; ANGLE 51.0 (Not valid for Circ layers and non-tubes)
$APO.CDIS=85
$VEL_EXTAX[1]=100
FOR N_CYC=1 to 26
 LIN_REL {X  -1.263,Y -17.738,A +0.664,E1 +5.909,E3 +39.726,E4 +39.726} C_DIS
 LIN_REL {X  -1.207,Y -17.519,A +6.151,E1 +1.101,E3 +33.522,E4 +33.522} C_DIS
 LIN_REL {X  +0.132,Y -25.137,A +10.003,E1 -0.421,E3 +50.269,E4 +50.269} C_DIS
 LIN_REL {X  +1.938,Y -24.469,A +9.586,E1 -2.860,E3 +55.196,E4 +55.196} C_DIS
 LIN_REL {X  +1.088,Y -27.792,A +3.019,E1 -0.955,E3 +68.896,E4 +68.896} C_DIS
 LIN_REL {X  -1.412,Y -27.938,A +0.462,E1 -0.637,E3 +74.120,E4 +74.120} C_DIS
 LIN_REL {X  -1.550,Y -28.084,A +0.079,E1 -0.824,E3 +75.675,E4 +75.675} C_DIS
 LIN_REL {X  -0.218,Y -37.855,A +0.031,E1 +0.120,E3 +99.590,E4 +99.590} C_DIS
 LIN_REL {X  +0.045,Y -439.757,A +0.006,E1 -0.006,E3 +1160.946,E4 +1160.946} C_DIS
 LIN_REL {X  -0.042,Y -41.169,A +0.005,E1 -0.034,E3 +108.768,E4 +108.768} C_DIS
 LIN_REL {X  +1.080,Y -35.595,A +0.045,E1 +0.289,E3 +92.600,E4 +92.600} C_DIS
 LIN_REL {X  +3.273,Y -34.380,A +0.217,E1 +0.416,E3 +91.278,E4 +91.278} C_DIS
 LIN_REL {X  +2.743,Y -26.470,A +1.240,E1 -2.201,E3 +76.331,E4 +76.331} C_DIS
 LIN_REL {X  +2.631,Y -16.478,A +6.378,E1 -6.830,E3 +59.126,E4 +59.126} C_DIS
 LIN_REL {X  +2.229,Y -8.399,A +11.491,E1 -13.235,E3 +51.842,E4 +51.842} C_DIS
 LIN_REL {X  +0.487,Y -0.700,A +8.521,E1 -13.721,E3 +42.558,E4 +42.558} C_DIS
 LIN_REL {X  -1.738,Y +4.804,A +2.101,E1 -9.621,E3 +38.319,E4 +38.319} C_DIS
 LIN_REL {X  -4.726,Y +16.117,A +0.001,E1 -12.271,E3 +54.688,E4 +54.688} C_DIS
 LIN_REL {X  -3.801,Y +19.459,A -0.092,E1 -8.574,E3 +43.826,E4 +43.826} C_DIS
 LIN_REL {X  -1.602,Y +15.638,A -4.416,E1 -2.235,E3 +29.939,E4 +29.939} C_DIS
 LIN_REL {X  -0.782,Y +22.587,A -8.423,E1 -0.320,E3 +44.108,E4 +44.108} C_DIS
 LIN_REL {X  +1.659,Y +27.200,A -11.255,E1 +2.496,E3 +59.206,E4 +59.206} C_DIS
 LIN_REL {X  +1.774,Y +29.070,A -4.803,E1 +1.404,E3 +70.515,E4 +70.515} C_DIS
 LIN_REL {X  -1.281,Y +30.779,A -0.863,E1 +0.755,E3 +80.640,E4 +80.640} C_DIS
 LIN_REL {X  -1.562,Y +27.869,A -0.109,E1 +1.005,E3 +75.559,E4 +75.559} C_DIS
 LIN_REL {X  -0.402,Y +34.896,A -0.035,E1 -0.167,E3 +91.664,E4 +91.664} C_DIS
 LIN_REL {X  +0.061,Y +446.163,A -0.005,E1 +0.005,E3 +1177.603,E4 +1177.603} C_DIS
 LIN_REL {X  -0.041,Y +41.178,A -0.009,E1 +0.036,E3 +108.772,E4 +108.772} C_DIS
 LIN_REL {X  +1.058,Y +35.617,A -0.046,E1 -0.293,E3 +92.627,E4 +92.627} C_DIS
 LIN_REL {X  +3.023,Y +32.120,A -0.168,E1 -0.412,E3 +85.081,E4 +85.081} C_DIS
 LIN_REL {X  +2.606,Y +25.937,A -0.789,E1 +1.529,E3 +73.528,E4 +73.528} C_DIS
 LIN_REL {X  +2.648,Y +17.147,A -4.931,E1 +5.567,E3 +58.465,E4 +58.465} C_DIS
 LIN_REL {X  +2.311,Y +9.487,A -12.018,E1 +12.736,E3 +50.262,E4 +50.262} C_DIS
 LIN_REL {X  +0.814,Y +2.053,A -9.484,E1 +14.819,E3 +47.597,E4 +47.597} C_DIS
 LIN_REL {X  -1.900,Y -4.606,A -2.553,E1 +10.763,E3 +43.244,E4 +43.244} C_DIS
 LIN_REL {X  -4.922,Y -13.188,A -0.001,E1 +10.333,E3 +35.563,E4 +35.563} C_DIS
 LIN_REL {X  -3.151,Y -10.847,A -0.000,E1 +6.334,E3 +35.274,E4 +35.274} C_DIS
ENDFOR

HALT
LIN {X -171.700,Y 1348.990,Z 0.000,A -27.171, B 0.00, C 0.00,E1 30.065}
HALT

; PLY 29 OF 41 (Connector)

; ANGLE 51.0 (Not valid for Circ layers and non-tubes)
$APO.CDIS=85
$VEL_EXTAX[1]=100
FOR N_CYC=1 to 1
 LIN_REL {X  +0.000,Y -9.233,A +0.373,E1 +2.358,E3 +17.818,E4 +17.818} C_DIS
 LIN_REL {X  +0.000,Y -13.860,A -0.779,E1 +4.453,E3 +24.815,E4 +24.815} C_DIS
 LIN_REL {X  +0.000,Y -18.793,A +5.783,E1 +1.657,E3 +30.501,E4 +30.501} C_DIS
 LIN_REL {X  +0.000,Y -28.514,A +11.207,E1 -0.369,E3 +47.105,E4 +47.105} C_DIS
 LIN_REL {X  +0.000,Y -29.574,A +8.105,E1 -0.986,E3 +52.158,E4 +52.158} C_DIS
 LIN_REL {X  +0.000,Y -39.267,A +2.075,E1 +1.140,E3 +70.967,E4 +70.967} C_DIS
 LIN_REL {X  +0.000,Y -46.416,A +0.339,E1 +1.591,E3 +81.647,E4 +81.647} C_DIS
 LIN_REL {X  +0.000,Y -56.639,A +0.061,E1 +2.018,E3 +93.300,E4 +93.300} C_DIS
 LIN_REL {X  +0.000,Y -63.527,A +0.007,E1 +2.194,E3 +97.039,E4 +97.039} C_DIS
 LIN_REL {X  +0.000,Y -66.959,A +0.000,E1 +2.174,E3 +94.666,E4 +94.666} C_DIS
 LIN_REL {X  +0.000,Y -70.250,A +0.000,E1 +2.135,E3 +91.980,E4 +91.980} C_DIS
 LIN_REL {X  +0.000,Y -70.396,A +0.000,E1 +2.009,E3 +85.511,E4 +85.511} C_DIS
 LIN_REL {X  +0.000,Y -73.804,A +0.000,E1 +1.984,E3 +83.251,E4 +83.251} C_DIS
 LIN_REL {X  +0.000,Y -77.291,A +0.000,E1 +1.961,E3 +80.882,E4 +80.882} C_DIS
 LIN_REL {X  +0.000,Y -77.374,A +0.002,E1 +1.847,E3 +75.125,E4 +75.125} C_DIS
 LIN_REL {X  +0.000,Y -70.709,A +0.068,E1 +1.551,E3 +64.105,E4 +64.105} C_DIS
 LIN_REL {X  +0.000,Y -55.789,A +0.709,E1 +0.995,E3 +48.959,E4 +48.959} C_DIS
 LIN_REL {X  +0.000,Y -40.604,A +4.575,E1 -1.183,E3 +41.358,E4 +41.358} C_DIS
 LIN_REL {X  +0.000,Y -25.454,A +10.692,E1 -5.269,E3 +34.062,E4 +34.062} C_DIS
 LIN_REL {X  +0.000,Y -12.708,A +10.798,E1 -8.471,E3 +24.267,E4 +24.267} C_DIS
 LIN_REL {X  +0.000,Y -7.379,A +3.152,E1 -5.505,E3 +25.747,E4 +25.747} C_DIS
 LIN_REL {X  +0.000,Y +0.970,A +0.004,E1 -4.558,E3 +33.819,E4 +33.819} C_DIS
 LIN_REL {X  +0.000,Y +10.934,A +0.000,E1 -10.007,E3 +28.863,E4 +28.863} C_DIS
 LIN_REL {X  +0.000,Y +19.588,A +0.000,E1 -13.423,E3 +28.165,E4 +28.165} C_DIS
 LIN_REL {X  +0.000,Y +12.206,A +0.000,E1 -10.399,E3 +11.631,E4 +11.631} C_DIS
 LIN_REL {X  +0.000,Y +1.140,A +0.000,E1 +0.761,E3 +0.965,E4 +0.965} C_DIS
 LIN_REL {X  +0.000,Y +3.435,A +0.000,E1 +4.724,E3 +3.121,E4 +3.121} C_DIS
 LIN_REL {X  +0.000,Y +16.386,A +0.000,E1 -14.565,E3 +13.019,E4 +13.019} C_DIS
 LIN_REL {X  +0.000,Y +31.237,A +0.000,E1 -16.911,E3 +19.850,E4 +19.850} C_DIS
 LIN_REL {X  +0.000,Y +24.263,A +0.000,E1 -12.079,E3 +15.482,E4 +15.482} C_DIS
ENDFOR

HALT
LIN {X -157.685,Y 535.549,Z 0.000,A 30.000, B 0.00, C 0.00,E1 -43.006}
HALT

; PLY 30 OF 41 (Helical)

; ANGLE 51.0 (Not valid for Circ layers and non-tubes)
$APO.CDIS=85
$VEL_EXTAX[1]=100
FOR N_CYC=1 to 49
 LIN_REL {X  -9.992,Y +38.440,A +0.000,E1 -12.506,E3 +27.076,E4 +27.076} C_DIS
 LIN_REL {X  -2.820,Y +34.329,A -0.140,E1 -4.875,E3 +21.050,E4 +21.050} C_DIS
 LIN_REL {X  -0.513,Y +17.919,A -5.095,E1 +0.029,E3 +11.726,E4 +11.726} C_DIS
 LIN_REL {X  -0.353,Y +14.948,A -0.644,E1 -0.565,E3 +10.215,E4 +10.215} C_DIS
 LIN_REL {X  -0.076,Y +14.598,A -1.861,E1 -0.455,E3 +10.433,E4 +10.433} C_DIS
 LIN_REL {X  +0.253,Y +25.054,A -7.468,E1 +0.260,E3 +18.780,E4 +18.780} C_DIS
 LIN_REL {X  +0.495,Y +39.543,A -9.068,E1 +0.940,E3 +31.936,E4 +31.936} C_DIS
 LIN_REL {X  +0.350,Y +52.493,A -5.061,E1 +0.537,E3 +46.398,E4 +46.398} C_DIS
 LIN_REL {X  +0.714,Y +65.315,A -0.637,E1 -0.061,E3 +60.775,E4 +60.775} C_DIS
 LIN_REL {X  +0.354,Y +72.797,A -0.026,E1 +0.019,E3 +68.477,E4 +68.477} C_DIS
 LIN_REL {X  +0.057,Y +276.942,A -0.000,E1 +0.012,E3 +261.192,E4 +261.192} C_DIS
 LIN_REL {X  +0.037,Y +57.440,A -0.000,E1 +0.014,E3 +54.220,E4 +54.220} C_DIS
 LIN_REL {X  +0.274,Y +42.150,A -0.000,E1 +0.085,E3 +40.041,E4 +40.041} C_DIS
 LIN_REL {X  +0.902,Y +29.530,A -0.002,E1 +0.226,E3 +28.682,E4 +28.682} C_DIS
 LIN_REL {X  +1.263,Y +17.565,A -0.005,E1 +0.283,E3 +17.684,E4 +17.684} C_DIS
 LIN_REL {X  +3.157,Y +23.364,A -0.024,E1 +0.665,E3 +24.764,E4 +24.764} C_DIS
 LIN_REL {X  +9.310,Y +31.543,A -0.347,E1 +1.862,E3 +37.286,E4 +37.286} C_DIS
 LIN_REL {X  +12.432,Y +18.699,A -3.734,E1 +3.126,E3 +27.471,E4 +27.471} C_DIS
 LIN_REL {X  +13.471,Y +12.237,A -11.704,E1 +6.647,E3 +27.002,E4 +27.002} C_DIS
 LIN_REL {X  +8.296,Y +6.142,A -8.436,E1 +5.968,E3 +20.449,E4 +20.449} C_DIS
 LIN_REL {X  +6.939,Y +4.164,A -2.979,E1 +4.722,E3 +22.940,E4 +22.940} C_DIS
 LIN_REL {X  +6.923,Y +3.493,A -2.751,E1 +10.488,E3 +42.442,E4 +42.442} C_DIS
 LIN_REL {X  -1.399,Y -0.415,A -0.018,E1 +13.616,E3 +55.399,E4 +55.399} C_DIS
 LIN_REL {X  -10.123,Y -6.481,A +0.000,E1 +15.056,E3 +45.794,E4 +45.794} C_DIS
 LIN_REL {X  -18.030,Y -13.565,A +0.000,E1 +18.431,E3 +41.692,E4 +41.692} C_DIS
 LIN_REL {X  -18.339,Y -23.904,A +0.000,E1 +18.670,E3 +32.802,E4 +32.802} C_DIS
 LIN_REL {X  -11.143,Y -31.247,A +0.000,E1 +12.210,E3 +24.387,E4 +24.387} C_DIS
 LIN_REL {X  -4.894,Y -37.209,A +0.000,E1 +7.145,E3 +22.801,E4 +22.801} C_DIS
 LIN_REL {X  -0.708,Y -20.875,A +2.543,E1 +0.987,E3 +13.371,E4 +13.371} C_DIS
 LIN_REL {X  -0.360,Y -13.653,A +4.268,E1 -0.155,E3 +9.150,E4 +9.150} C_DIS
 LIN_REL {X  -0.243,Y -17.021,A -0.267,E1 +0.899,E3 +11.930,E4 +11.930} C_DIS
 LIN_REL {X  +0.170,Y -22.146,A +6.338,E1 -0.020,E3 +16.273,E4 +16.273} C_DIS
 LIN_REL {X  +0.520,Y -34.300,A +8.556,E1 -0.682,E3 +26.945,E4 +26.945} C_DIS
 LIN_REL {X  +0.275,Y -48.825,A +7.263,E1 -0.966,E3 +42.019,E4 +42.019} C_DIS
 LIN_REL {X  +0.615,Y -59.709,A +1.212,E1 +0.086,E3 +55.054,E4 +55.054} C_DIS
 LIN_REL {X  +0.533,Y -71.084,A +0.084,E1 -0.000,E3 +66.733,E4 +66.733} C_DIS
 LIN_REL {X  +0.122,Y -305.348,A +0.003,E1 -0.022,E3 +287.956,E4 +287.956} C_DIS
 LIN_REL {X  +0.045,Y -57.401,A +0.000,E1 -0.017,E3 +54.194,E4 +54.194} C_DIS
 LIN_REL {X  +0.339,Y -41.950,A +0.000,E1 -0.101,E3 +39.910,E4 +39.910} C_DIS
 LIN_REL {X  +1.030,Y -29.366,A +0.002,E1 -0.250,E3 +28.637,E4 +28.637} C_DIS
 LIN_REL {X  +1.070,Y -14.362,A +0.003,E1 -0.238,E3 +14.492,E4 +14.492} C_DIS
 LIN_REL {X  +2.587,Y -20.443,A +0.016,E1 -0.547,E3 +21.523,E4 +21.523} C_DIS
 LIN_REL {X  +7.682,Y -29.414,A +0.236,E1 -1.546,E3 +34.044,E4 +34.044} C_DIS
 LIN_REL {X  +11.916,Y -20.738,A +2.572,E1 -2.756,E3 +28.891,E4 +28.891} C_DIS
 LIN_REL {X  +13.331,Y -12.978,A +10.132,E1 -5.754,E3 +26.094,E4 +26.094} C_DIS
 LIN_REL {X  +10.908,Y -8.239,A +10.945,E1 -7.427,E3 +25.783,E4 +25.783} C_DIS
 LIN_REL {X  +8.205,Y -4.895,A +3.479,E1 -5.602,E3 +27.304,E4 +27.304} C_DIS
 LIN_REL {X  +5.935,Y -2.966,A +2.598,E1 -9.964,E3 +39.224,E4 +39.224} C_DIS
 LIN_REL {X  -1.496,Y +0.449,A +0.017,E1 -13.553,E3 +55.117,E4 +55.117} C_DIS
 LIN_REL {X  -10.127,Y +6.477,A +0.000,E1 -14.993,E3 +45.594,E4 +45.594} C_DIS
 LIN_REL {X  -17.619,Y +12.986,A +0.000,E1 -18.049,E3 +40.676,E4 +40.676} C_DIS
 LIN_REL {X  -22.275,Y +29.917,A +0.000,E1 -21.879,E3 +38.845,E4 +38.845} C_DIS
ENDFOR

HALT
LIN {X -172.144,Y 529.033,Z 0.000,A 30.000, B 0.00, C 0.00,E1 -44.225}
HALT

; PLY 31 OF 41 (Connector)

; ANGLE 51.0 (Not valid for Circ layers and non-tubes)
$APO.CDIS=85
$VEL_EXTAX[1]=100
FOR N_CYC=1 to 1
 LIN_REL {X  +0.000,Y +14.319,A +0.000,E1 -4.145,E3 +12.342,E4 +12.342} C_DIS
 LIN_REL {X  +0.000,Y +6.169,A +0.000,E1 -1.493,E3 +5.195,E4 +5.195} C_DIS
 LIN_REL {X  +0.000,Y +13.714,A +0.000,E1 -3.208,E3 +10.742,E4 +10.742} C_DIS
 LIN_REL {X  +0.000,Y +36.143,A -0.001,E1 -5.463,E3 +24.130,E4 +24.130} C_DIS
 LIN_REL {X  +0.000,Y +26.736,A -3.446,E1 -0.505,E3 +19.551,E4 +19.551} C_DIS
 LIN_REL {X  +0.000,Y +25.698,A -6.360,E1 +0.299,E3 +22.076,E4 +22.076} C_DIS
 LIN_REL {X  +0.000,Y +35.270,A -10.863,E1 +1.539,E3 +33.206,E4 +33.206} C_DIS
 LIN_REL {X  +0.000,Y +38.420,A -7.659,E1 +2.559,E3 +44.300,E4 +44.300} C_DIS
 LIN_REL {X  +0.000,Y +44.211,A -1.519,E1 +1.891,E3 +58.868,E4 +58.868} C_DIS
 LIN_REL {X  +0.000,Y +49.956,A -0.142,E1 +1.911,E3 +70.742,E4 +70.742} C_DIS
 LIN_REL {X  +0.000,Y +56.506,A -0.010,E1 +2.198,E3 +85.749,E4 +85.749} C_DIS
 LIN_REL {X  +0.000,Y +61.033,A +0.000,E1 +2.498,E3 +100.307,E4 +100.307} C_DIS
 LIN_REL {X  +0.000,Y +58.632,A +0.000,E1 +2.584,E3 +105.218,E4 +105.218} C_DIS
 LIN_REL {X  +0.000,Y +53.534,A -0.000,E1 +2.555,E3 +105.199,E4 +105.199} C_DIS
 LIN_REL {X  +0.000,Y +41.233,A -0.000,E1 +2.127,E3 +88.197,E4 +88.197} C_DIS
 LIN_REL {X  +0.000,Y +31.694,A -0.000,E1 +1.788,E3 +72.960,E4 +72.960} C_DIS
 LIN_REL {X  +0.000,Y +22.339,A -0.000,E1 +1.883,E3 +54.647,E4 +54.647} C_DIS
 LIN_REL {X  +0.000,Y +12.026,A -0.000,E1 +1.596,E3 +30.477,E4 +30.477} C_DIS
 LIN_REL {X  +0.000,Y +8.605,A -0.000,E1 +0.479,E3 +23.899,E4 +23.899} C_DIS
 LIN_REL {X  +0.000,Y +17.185,A -0.000,E1 +0.297,E3 +43.997,E4 +43.997} C_DIS
 LIN_REL {X  +0.000,Y +22.397,A -0.002,E1 +1.554,E3 +63.484,E4 +63.484} C_DIS
 LIN_REL {X  +0.000,Y +26.340,A -0.006,E1 +1.986,E3 +80.445,E4 +80.445} C_DIS
 LIN_REL {X  +0.000,Y +29.797,A -0.026,E1 +2.502,E3 +100.345,E4 +100.345} C_DIS
 LIN_REL {X  +0.000,Y +26.761,A -0.089,E1 +2.608,E3 +101.540,E4 +101.540} C_DIS
 LIN_REL {X  +0.000,Y +19.332,A -0.202,E1 +2.288,E3 +83.045,E4 +83.045} C_DIS
 LIN_REL {X  +0.000,Y +13.522,A -0.387,E1 +2.080,E3 +65.819,E4 +65.819} C_DIS
 LIN_REL {X  +0.000,Y +9.350,A -0.577,E1 +1.526,E3 +48.552,E4 +48.552} C_DIS
 LIN_REL {X  +0.000,Y +7.090,A -1.004,E1 +0.962,E3 +34.729,E4 +34.729} C_DIS
 LIN_REL {X  +0.000,Y +4.780,A -0.977,E1 +1.016,E3 +28.901,E4 +28.901} C_DIS
 LIN_REL {X  +0.000,Y +4.146,A -1.612,E1 +2.199,E3 +25.934,E4 +25.934} C_DIS
 LIN_REL {X  +0.000,Y +5.726,A -4.369,E1 +5.416,E3 +44.520,E4 +44.520} C_DIS
 LIN_REL {X  +0.000,Y +2.416,A -7.629,E1 +11.123,E3 +57.450,E4 +57.450} C_DIS
 LIN_REL {X  +0.000,Y -2.383,A -3.896,E1 +8.270,E3 +42.248,E4 +42.248} C_DIS
 LIN_REL {X  +0.000,Y -1.687,A -0.589,E1 +2.742,E3 +18.919,E4 +18.919} C_DIS
ENDFOR

HALT
LIN {X -169.560,Y 1333.646,Z 0.000,A -22.240, B 0.00, C 0.00,E1 22.754}
HALT

; PLY 32 OF 41 (Helical)

; ANGLE 51.0 (Not valid for Circ layers and non-tubes)
$APO.CDIS=85
$VEL_EXTAX[1]=100
FOR N_CYC=1 to 16
 LIN_REL {X  +3.047,Y -12.617,A +5.110,E1 +1.887,E3 +50.457,E4 +50.457} C_DIS
 LIN_REL {X  +0.960,Y -17.440,A +9.214,E1 -2.081,E3 +64.163,E4 +64.163} C_DIS
 LIN_REL {X  -1.414,Y -14.583,A +4.594,E1 -1.524,E3 +56.231,E4 +56.231} C_DIS
 LIN_REL {X  -1.370,Y -15.018,A +2.113,E1 -0.735,E3 +62.283,E4 +62.283} C_DIS
 LIN_REL {X  -1.253,Y -19.133,A +0.727,E1 -0.124,E3 +82.087,E4 +82.087} C_DIS
 LIN_REL {X  -0.026,Y -22.209,A +0.320,E1 -0.224,E3 +98.503,E4 +98.503} C_DIS
 LIN_REL {X  +0.451,Y -26.687,A +0.109,E1 +0.014,E3 +118.641,E4 +118.641} C_DIS
 LIN_REL {X  +0.291,Y -27.443,A +0.036,E1 +0.011,E3 +122.245,E4 +122.245} C_DIS
 LIN_REL {X  +0.127,Y -27.130,A +0.012,E1 +0.006,E3 +120.899,E4 +120.899} C_DIS
 LIN_REL {X  +0.051,Y -411.402,A +0.005,E1 +0.000,E3 +1833.463,E4 +1833.463} C_DIS
 LIN_REL {X  -0.039,Y -28.657,A +0.002,E1 -0.012,E3 +127.754,E4 +127.754} C_DIS
 LIN_REL {X  -0.105,Y -27.141,A +0.010,E1 -0.033,E3 +121.065,E4 +121.065} C_DIS
 LIN_REL {X  -0.219,Y -26.340,A +0.034,E1 -0.084,E3 +117.665,E4 +117.665} C_DIS
 LIN_REL {X  -0.310,Y -25.741,A +0.107,E1 -0.189,E3 +115.235,E4 +115.235} C_DIS
 LIN_REL {X  +0.425,Y -23.022,A +0.379,E1 -0.330,E3 +102.988,E4 +102.988} C_DIS
 LIN_REL {X  +2.360,Y -18.319,A +0.615,E1 -0.563,E3 +85.228,E4 +85.228} C_DIS
 LIN_REL {X  +2.831,Y -12.780,A +2.165,E1 -2.874,E3 +73.426,E4 +73.426} C_DIS
 LIN_REL {X  +1.801,Y -7.188,A +3.504,E1 -5.269,E3 +62.055,E4 +62.055} C_DIS
 LIN_REL {X  -0.788,Y -1.801,A +7.426,E1 -11.611,E3 +62.049,E4 +62.049} C_DIS
 LIN_REL {X  -1.919,Y +4.462,A +3.832,E1 -9.497,E3 +52.182,E4 +52.182} C_DIS
 LIN_REL {X  -1.406,Y +8.884,A +1.558,E1 -7.940,E3 +51.827,E4 +51.827} C_DIS
 LIN_REL {X  -0.156,Y +13.630,A -2.139,E1 -4.967,E3 +55.231,E4 +55.231} C_DIS
 LIN_REL {X  +0.635,Y +14.690,A -6.813,E1 -0.035,E3 +54.948,E4 +54.948} C_DIS
 LIN_REL {X  -0.874,Y +16.392,A -6.472,E1 +2.299,E3 +62.626,E4 +62.626} C_DIS
 LIN_REL {X  -1.522,Y +14.707,A -2.530,E1 +0.595,E3 +59.944,E4 +59.944} C_DIS
 LIN_REL {X  -1.416,Y +18.139,A -1.020,E1 +0.294,E3 +76.766,E4 +76.766} C_DIS
 LIN_REL {X  -0.288,Y +21.343,A -0.419,E1 +0.247,E3 +94.415,E4 +94.415} C_DIS
 LIN_REL {X  +0.419,Y +26.139,A -0.172,E1 +0.022,E3 +116.135,E4 +116.135} C_DIS
 LIN_REL {X  +0.342,Y +27.112,A -0.049,E1 -0.009,E3 +120.665,E4 +120.665} C_DIS
 LIN_REL {X  +0.161,Y +28.178,A -0.014,E1 -0.009,E3 +125.507,E4 +125.507} C_DIS
 LIN_REL {X  +0.069,Y +417.342,A -0.005,E1 -0.002,E3 +1859.921,E4 +1859.921} C_DIS
 LIN_REL {X  -0.039,Y +28.657,A -0.004,E1 +0.013,E3 +127.755,E4 +127.755} C_DIS
 LIN_REL {X  -0.104,Y +27.140,A -0.011,E1 +0.034,E3 +121.066,E4 +121.066} C_DIS
 LIN_REL {X  -0.222,Y +26.341,A -0.033,E1 +0.083,E3 +117.668,E4 +117.668} C_DIS
 LIN_REL {X  -0.326,Y +25.743,A -0.094,E1 +0.178,E3 +115.235,E4 +115.235} C_DIS
 LIN_REL {X  +0.389,Y +23.022,A -0.321,E1 +0.285,E3 +102.960,E4 +102.960} C_DIS
 LIN_REL {X  +2.313,Y +18.360,A -0.543,E1 +0.478,E3 +84.986,E4 +84.986} C_DIS
 LIN_REL {X  +3.085,Y +13.902,A -2.268,E1 +2.948,E3 +79.333,E4 +79.333} C_DIS
 LIN_REL {X  +1.875,Y +6.705,A -4.011,E1 +5.854,E3 +60.866,E4 +60.866} C_DIS
 LIN_REL {X  -1.178,Y +1.377,A -8.203,E1 +12.683,E3 +62.451,E4 +62.451} C_DIS
 LIN_REL {X  -3.235,Y -4.878,A -4.375,E1 +9.532,E3 +39.515,E4 +39.515} C_DIS
 LIN_REL {X  -2.005,Y -5.975,A -1.476,E1 +5.423,E3 +17.981,E4 +17.981} C_DIS
 LIN_REL {X  -1.418,Y -6.761,A -0.900,E1 +5.226,E3 +51.080,E4 +51.080} C_DIS
ENDFOR

HALT
LIN {X -172.581,Y 1334.232,Z 0.000,A -8.411, B 0.00, C 0.00,E1 12.625}
HALT

; PLY 33 OF 41 (Connector)

; ANGLE 51.0 (Not valid for Circ layers and non-tubes)
$APO.CDIS=85
$VEL_EXTAX[1]=100
FOR N_CYC=1 to 1
 LIN_REL {X  +0.000,Y -5.046,A -0.366,E1 +2.248,E3 +23.242,E4 +23.242} C_DIS
 LIN_REL {X  +0.000,Y -7.414,A -1.041,E1 +3.480,E3 +33.385,E4 +33.385} C_DIS
 LIN_REL {X  +0.000,Y -10.497,A -0.806,E1 +4.034,E3 +33.290,E4 +33.290} C_DIS
 LIN_REL {X  +0.000,Y -19.865,A +4.800,E1 +1.630,E3 +57.784,E4 +57.784} C_DIS
 LIN_REL {X  +0.000,Y -29.613,A +4.205,E1 +1.810,E3 +79.851,E4 +79.851} C_DIS
 LIN_REL {X  +0.000,Y -39.427,A +1.225,E1 +3.725,E3 +93.792,E4 +93.792} C_DIS
 LIN_REL {X  +0.000,Y -50.165,A +0.317,E1 +4.475,E3 +102.300,E4 +102.300} C_DIS
 LIN_REL {X  +0.000,Y -55.940,A +0.066,E1 +4.406,E3 +97.463,E4 +97.463} C_DIS
 LIN_REL {X  +0.000,Y -63.480,A +0.010,E1 +4.376,E3 +94.812,E4 +94.812} C_DIS
 LIN_REL {X  +0.000,Y -67.312,A +0.001,E1 +4.069,E3 +86.665,E4 +86.665} C_DIS
 LIN_REL {X  +0.000,Y -75.350,A +0.000,E1 +4.013,E3 +83.734,E4 +83.734} C_DIS
 LIN_REL {X  +0.000,Y -78.546,A +0.000,E1 +3.712,E3 +75.243,E4 +75.243} C_DIS
 LIN_REL {X  +0.000,Y -83.487,A +0.000,E1 +3.528,E3 +68.787,E4 +68.787} C_DIS
 LIN_REL {X  +0.000,Y -89.192,A +0.000,E1 +3.382,E3 +62.739,E4 +62.739} C_DIS
 LIN_REL {X  +0.000,Y -91.855,A +0.003,E1 +3.131,E3 +54.649,E4 +54.649} C_DIS
 LIN_REL {X  +0.000,Y -89.044,A +0.052,E1 +2.725,E3 +44.748,E4 +44.748} C_DIS
 LIN_REL {X  +0.000,Y -71.953,A +0.418,E1 +1.912,E3 +32.096,E4 +32.096} C_DIS
 LIN_REL {X  +0.000,Y -55.976,A +1.865,E1 +0.621,E3 +28.664,E4 +28.664} C_DIS
 LIN_REL {X  +0.000,Y -39.642,A +4.492,E1 -0.776,E3 +26.538,E4 +26.538} C_DIS
 LIN_REL {X  +0.000,Y -23.550,A +5.744,E1 -1.723,E3 +18.264,E4 +18.264} C_DIS
 LIN_REL {X  +0.000,Y -13.214,A +1.694,E1 +1.653,E3 +16.607,E4 +16.607} C_DIS
 LIN_REL {X  +0.000,Y -10.967,A +6.864,E1 -2.996,E3 +23.427,E4 +23.427} C_DIS
 LIN_REL {X  +0.000,Y -7.196,A +7.994,E1 -8.065,E3 +40.118,E4 +40.118} C_DIS
 LIN_REL {X  +0.000,Y +10.943,A +0.873,E1 -5.390,E3 +39.498,E4 +39.498} C_DIS
 LIN_REL {X  +0.000,Y +12.495,A +0.001,E1 -5.685,E3 +16.816,E4 +16.816} C_DIS
 LIN_REL {X  +0.000,Y +5.972,A +0.000,E1 -5.914,E3 +6.076,E4 +6.076} C_DIS
 LIN_REL {X  +0.000,Y -8.713,A +0.000,E1 +14.347,E3 +0.236,E4 +0.236} C_DIS
 LIN_REL {X  +0.000,Y -2.670,A +0.000,E1 +1.637,E3 +0.118,E4 +0.118} C_DIS
 LIN_REL {X  +0.000,Y +12.391,A +0.000,E1 -7.123,E3 +7.454,E4 +7.454} C_DIS
 LIN_REL {X  +0.000,Y +40.457,A +0.000,E1 -13.567,E3 +27.870,E4 +27.870} C_DIS
 LIN_REL {X  +0.000,Y +25.086,A +0.000,E1 -11.150,E3 +13.685,E4 +13.685} C_DIS
 LIN_REL {X  +0.000,Y +10.925,A +0.000,E1 -2.042,E3 +5.363,E4 +5.363} C_DIS
 LIN_REL {X  +0.000,Y +11.929,A +0.000,E1 +1.715,E3 +5.191,E4 +5.191} C_DIS
 LIN_REL {X  +0.000,Y +12.060,A +0.000,E1 -8.475,E3 +4.873,E4 +4.873} C_DIS
 LIN_REL {X  +0.000,Y +18.561,A +0.000,E1 -14.986,E3 +7.188,E4 +7.188} C_DIS
 LIN_REL {X  +0.000,Y +11.788,A +0.000,E1 -7.556,E3 +4.362,E4 +4.362} C_DIS
 LIN_REL {X  +0.000,Y +3.641,A +0.000,E1 -0.711,E3 +1.727,E4 +1.727} C_DIS
 LIN_REL {X  +0.000,Y +4.304,A +0.000,E1 +0.673,E3 +3.439,E4 +3.439} C_DIS
 LIN_REL {X  +0.000,Y +17.578,A +0.000,E1 -10.494,E3 +5.358,E4 +5.358} C_DIS
 LIN_REL {X  +0.000,Y +28.849,A +0.000,E1 -19.404,E3 +7.468,E4 +7.468} C_DIS
 LIN_REL {X  +0.000,Y +24.716,A +0.000,E1 -13.059,E3 +5.156,E4 +5.156} C_DIS
 LIN_REL {X  +0.000,Y +7.033,A +0.000,E1 -2.445,E3 +1.952,E4 +1.952} C_DIS
 LIN_REL {X  +0.000,Y -7.825,A +0.000,E1 +3.615,E3 +4.095,E4 +4.095} C_DIS
 LIN_REL {X  +0.000,Y +12.443,A +0.000,E1 -4.870,E3 +9.533,E4 +9.533} C_DIS
 LIN_REL {X  +0.000,Y +11.720,A +0.000,E1 -2.877,E3 +7.487,E4 +7.487} C_DIS
 LIN_REL {X  +0.000,Y +9.258,A +0.000,E1 -2.259,E3 +5.089,E4 +5.089} C_DIS
 LIN_REL {X  +0.000,Y +9.556,A +0.000,E1 -2.180,E3 +4.911,E4 +4.911} C_DIS
 LIN_REL {X  +0.000,Y -3.275,A +0.000,E1 +0.940,E3 +2.074,E4 +2.074} C_DIS
 LIN_REL {X  +0.000,Y +17.086,A +0.000,E1 -5.772,E3 +3.326,E4 +3.326} C_DIS
 LIN_REL {X  +0.000,Y +23.595,A +0.000,E1 -2.897,E3 +5.507,E4 +5.507} C_DIS
 LIN_REL {X  +0.000,Y +9.529,A +0.000,E1 -1.296,E3 +2.945,E4 +2.945} C_DIS
 LIN_REL {X  +0.000,Y +31.401,A -0.001,E1 -2.087,E3 +9.384,E4 +9.384} C_DIS
 LIN_REL {X  +0.000,Y +24.719,A -2.524,E1 -0.136,E3 +8.548,E4 +8.548} C_DIS
 LIN_REL {X  +0.000,Y +5.465,A +0.374,E1 -0.017,E3 +2.890,E4 +2.890} C_DIS
 LIN_REL {X  +0.000,Y -4.461,A +0.964,E1 -0.970,E3 +0.620,E4 +0.620} C_DIS
 LIN_REL {X  +0.000,Y +19.335,A -6.127,E1 +0.144,E3 +6.624,E4 +6.624} C_DIS
 LIN_REL {X  +0.000,Y +38.084,A -9.162,E1 +0.108,E3 +15.408,E4 +15.408} C_DIS
 LIN_REL {X  +0.000,Y +37.799,A -6.128,E1 +1.334,E3 +15.871,E4 +15.871} C_DIS
 LIN_REL {X  +0.000,Y +25.082,A +0.780,E1 -1.223,E3 +10.271,E4 +10.271} C_DIS
 LIN_REL {X  +0.000,Y +31.070,A -3.297,E1 +0.126,E3 +13.286,E4 +13.286} C_DIS
 LIN_REL {X  +0.000,Y +48.551,A -3.056,E1 +0.056,E3 +21.505,E4 +21.505} C_DIS
 LIN_REL {X  +0.000,Y +66.788,A -1.592,E1 -0.126,E3 +31.712,E4 +31.712} C_DIS
 LIN_REL {X  +0.000,Y +80.524,A -0.224,E1 +0.020,E3 +40.557,E4 +40.557} C_DIS
 LIN_REL {X  +0.000,Y +322.024,A -0.007,E1 +0.007,E3 +162.586,E4 +162.586} C_DIS
 LIN_REL {X  +0.000,Y +97.753,A -0.002,E1 +0.001,E3 +49.360,E4 +49.360} C_DIS
 LIN_REL {X  +0.000,Y +78.475,A -0.060,E1 +0.015,E3 +39.653,E4 +39.653} C_DIS
 LIN_REL {X  +0.000,Y +60.129,A -0.527,E1 +0.034,E3 +30.613,E4 +30.613} C_DIS
 LIN_REL {X  +0.000,Y +45.249,A -2.028,E1 +0.080,E3 +24.217,E4 +24.217} C_DIS
 LIN_REL {X  +0.000,Y +32.360,A -3.378,E1 +0.393,E3 +19.311,E4 +19.311} C_DIS
 LIN_REL {X  +0.000,Y +14.965,A -2.298,E1 +0.414,E3 +9.799,E4 +9.799} C_DIS
 LIN_REL {X  +0.000,Y +19.479,A -3.937,E1 +0.978,E3 +13.776,E4 +13.776} C_DIS
 LIN_REL {X  +0.000,Y +22.145,A -4.242,E1 +1.224,E3 +18.263,E4 +18.263} C_DIS
 LIN_REL {X  +0.000,Y +11.110,A -5.497,E1 -0.418,E3 +20.566,E4 +20.566} C_DIS
 LIN_REL {X  +0.000,Y +6.860,A -6.486,E1 +4.424,E3 +24.845,E4 +24.845} C_DIS
 LIN_REL {X  +0.000,Y -2.704,A -1.542,E1 +5.717,E3 +43.329,E4 +43.329} C_DIS
 LIN_REL {X  +0.000,Y -22.047,A -0.003,E1 +5.153,E3 +37.053,E4 +37.053} C_DIS
 LIN_REL {X  +0.000,Y -15.523,A +0.000,E1 +8.983,E3 +12.765,E4 +12.765} C_DIS
 LIN_REL {X  +0.000,Y +0.049,A +0.000,E1 +0.761,E3 +1.038,E4 +1.038} C_DIS
 LIN_REL {X  +0.000,Y +10.478,A +0.000,E1 -14.571,E3 +0.837,E4 +0.837} C_DIS
 LIN_REL {X  +0.000,Y +3.006,A +0.000,E1 -1.717,E3 +0.418,E4 +0.418} C_DIS
 LIN_REL {X  +0.000,Y -13.163,A +0.000,E1 +6.413,E3 +3.779,E4 +3.779} C_DIS
 LIN_REL {X  +0.000,Y -35.643,A +0.000,E1 +9.685,E3 +21.819,E4 +21.819} C_DIS
 LIN_REL {X  +0.000,Y -38.214,A +0.000,E1 +13.732,E3 +18.951,E4 +18.951} C_DIS
 LIN_REL {X  +0.000,Y -16.826,A +0.000,E1 +3.973,E3 +7.217,E4 +7.217} C_DIS
 LIN_REL {X  +0.000,Y -13.110,A +0.000,E1 -2.140,E3 +4.897,E4 +4.897} C_DIS
 LIN_REL {X  +0.000,Y -12.296,A +0.000,E1 +8.348,E3 +4.340,E4 +4.340} C_DIS
 LIN_REL {X  +0.000,Y -21.267,A +0.000,E1 +17.266,E3 +7.205,E4 +7.205} C_DIS
 LIN_REL {X  +0.000,Y -14.448,A +0.000,E1 +8.473,E3 +4.704,E4 +4.704} C_DIS
 LIN_REL {X  +0.000,Y -0.703,A +0.000,E1 -0.558,E3 +0.489,E4 +0.489} C_DIS
 LIN_REL {X  +0.000,Y -2.667,A +0.000,E1 -2.696,E3 +2.537,E4 +2.537} C_DIS
 LIN_REL {X  +0.000,Y -14.072,A +0.000,E1 +8.194,E3 +3.863,E4 +3.863} C_DIS
 LIN_REL {X  +0.000,Y -24.341,A +0.000,E1 +19.073,E3 +6.002,E4 +6.002} C_DIS
 LIN_REL {X  +0.000,Y -34.103,A +0.000,E1 +19.291,E3 +6.792,E4 +6.792} C_DIS
 LIN_REL {X  +0.000,Y -12.687,A +0.000,E1 +5.644,E3 +2.011,E4 +2.011} C_DIS
 LIN_REL {X  +0.000,Y +15.588,A +0.000,E1 -10.283,E3 +0.478,E4 +0.478} C_DIS
 LIN_REL {X  +0.000,Y +1.851,A +0.000,E1 +0.107,E3 +0.096,E4 +0.096} C_DIS
 LIN_REL {X  +0.000,Y -19.694,A +0.000,E1 +9.999,E3 +12.329,E4 +12.329} C_DIS
ENDFOR

HALT
LIN {X -153.780,Y 1393.090,Z 0.000,A -30.000, B 0.00, C 0.00,E1 57.931}
HALT

; PLY 34 OF 41 (Helical)

; ANGLE 51.0 (Not valid for Circ layers and non-tubes)
$APO.CDIS=85
$VEL_EXTAX[1]=100
FOR N_CYC=1 to 57
 LIN_REL {X  -6.080,Y -11.205,A +0.000,E1 +3.668,E3 +9.842,E4 +9.842} C_DIS
 LIN_REL {X  -2.471,Y -7.290,A +0.000,E1 +1.453,E3 +6.006,E4 +6.006} C_DIS
 LIN_REL {X  -6.094,Y -25.471,A +0.000,E1 +5.807,E3 +7.774,E4 +7.774} C_DIS
 LIN_REL {X  -3.295,Y -38.249,A +0.000,E1 +3.173,E3 +12.247,E4 +12.247} C_DIS
 LIN_REL {X  -0.466,Y -19.876,A +2.308,E1 +0.082,E3 +7.015,E4 +7.015} C_DIS
 LIN_REL {X  -0.159,Y -12.565,A +2.013,E1 +0.203,E3 +4.588,E4 +4.588} C_DIS
 LIN_REL {X  +0.104,Y -14.761,A -1.934,E1 +0.802,E3 +5.522,E4 +5.522} C_DIS
 LIN_REL {X  +0.261,Y -21.215,A +7.084,E1 -0.128,E3 +8.127,E4 +8.127} C_DIS
 LIN_REL {X  +0.164,Y -30.530,A +10.070,E1 -0.732,E3 +12.002,E4 +12.002} C_DIS
 LIN_REL {X  -0.078,Y -26.825,A +2.365,E1 -0.215,E3 +10.811,E4 +10.811} C_DIS
 LIN_REL {X  -0.123,Y -35.256,A -0.737,E1 +0.491,E3 +14.704,E4 +14.704} C_DIS
 LIN_REL {X  +0.174,Y -46.272,A +4.747,E1 -0.178,E3 +20.444,E4 +20.444} C_DIS
 LIN_REL {X  -0.120,Y -64.963,A +3.362,E1 -0.233,E3 +30.616,E4 +30.616} C_DIS
 LIN_REL {X  +0.008,Y -78.909,A +0.685,E1 +0.042,E3 +39.385,E4 +39.385} C_DIS
 LIN_REL {X  +0.092,Y -105.486,A +0.037,E1 -0.014,E3 +53.242,E4 +53.242} C_DIS
 LIN_REL {X  +0.008,Y -111.830,A -0.000,E1 -0.002,E3 +56.484,E4 +56.484} C_DIS
 LIN_REL {X  +0.095,Y -75.413,A +0.000,E1 -0.012,E3 +38.165,E4 +38.165} C_DIS
 LIN_REL {X  +1.097,Y -60.416,A +0.000,E1 -0.126,E3 +31.379,E4 +31.379} C_DIS
 LIN_REL {X  +4.654,Y -45.960,A +0.000,E1 -0.515,E3 +26.730,E4 +26.730} C_DIS
 LIN_REL {X  +9.134,Y -28.884,A +0.007,E1 -1.051,E3 +20.983,E4 +20.983} C_DIS
 LIN_REL {X  +7.649,Y -12.781,A +0.066,E1 -0.946,E3 +11.193,E4 +11.193} C_DIS
 LIN_REL {X  +15.165,Y -16.332,A +2.567,E1 -2.232,E3 +15.876,E4 +15.876} C_DIS
 LIN_REL {X  +10.999,Y -8.398,A +4.811,E1 -2.014,E3 +10.197,E4 +10.197} C_DIS
 LIN_REL {X  +11.317,Y -7.162,A +3.067,E1 -2.479,E3 +12.051,E4 +12.051} C_DIS
 LIN_REL {X  +11.135,Y -6.819,A +11.749,E1 -4.816,E3 +15.427,E4 +15.427} C_DIS
 LIN_REL {X  +7.334,Y -5.384,A +6.253,E1 -3.915,E3 +13.866,E4 +13.866} C_DIS
 LIN_REL {X  +7.865,Y -11.086,A +0.565,E1 -3.452,E3 +25.588,E4 +25.588} C_DIS
 LIN_REL {X  +5.482,Y -19.357,A +0.908,E1 -4.733,E3 +47.099,E4 +47.099} C_DIS
 LIN_REL {X  -0.294,Y -15.438,A +0.007,E1 -10.306,E3 +66.498,E4 +66.498} C_DIS
 LIN_REL {X  -2.988,Y +5.027,A -0.000,E1 -9.870,E3 +44.670,E4 +44.670} C_DIS
 LIN_REL {X  -1.270,Y +20.815,A -0.000,E1 -14.160,E3 +34.085,E4 +34.085} C_DIS
 LIN_REL {X  -6.380,Y +17.426,A -0.000,E1 -11.604,E3 +26.837,E4 +26.837} C_DIS
 LIN_REL {X  -12.275,Y +10.982,A -0.000,E1 -17.052,E3 +22.453,E4 +22.453} C_DIS
 LIN_REL {X  -11.596,Y +8.222,A -0.000,E1 -13.757,E3 +14.467,E4 +14.467} C_DIS
 LIN_REL {X  -7.704,Y +4.618,A -0.000,E1 -5.069,E3 +8.828,E4 +8.828} C_DIS
 LIN_REL {X  -7.566,Y +4.986,A -0.000,E1 -5.000,E3 +12.964,E4 +12.964} C_DIS
 LIN_REL {X  -14.348,Y +14.863,A -0.000,E1 -11.439,E3 +17.644,E4 +17.644} C_DIS
 LIN_REL {X  -10.023,Y +13.413,A -0.000,E1 -6.426,E3 +12.228,E4 +12.228} C_DIS
 LIN_REL {X  -6.487,Y +10.519,A -0.000,E1 -2.992,E3 +8.976,E4 +8.976} C_DIS
 LIN_REL {X  -4.224,Y +15.376,A -0.000,E1 -3.977,E3 +6.193,E4 +6.193} C_DIS
 LIN_REL {X  -5.660,Y +35.371,A -0.000,E1 -4.970,E3 +10.726,E4 +10.726} C_DIS
 LIN_REL {X  -1.282,Y +32.472,A -0.472,E1 -1.464,E3 +11.027,E4 +11.027} C_DIS
 LIN_REL {X  -0.256,Y +14.504,A -3.684,E1 +0.065,E3 +5.245,E4 +5.245} C_DIS
 LIN_REL {X  -0.017,Y +11.804,A +2.076,E1 -0.686,E3 +4.380,E4 +4.380} C_DIS
 LIN_REL {X  +0.222,Y +17.165,A -3.176,E1 -0.330,E3 +6.522,E4 +6.522} C_DIS
 LIN_REL {X  +0.297,Y +31.207,A -10.805,E1 +0.602,E3 +12.175,E4 +12.175} C_DIS
 LIN_REL {X  -0.009,Y +28.214,A -6.569,E1 +0.610,E3 +11.297,E4 +11.297} C_DIS
 LIN_REL {X  -0.203,Y +29.676,A +1.200,E1 -0.226,E3 +12.191,E4 +12.191} C_DIS
 LIN_REL {X  -0.032,Y +35.676,A -1.670,E1 -0.380,E3 +15.316,E4 +15.316} C_DIS
 LIN_REL {X  +0.154,Y +53.398,A -4.669,E1 +0.379,E3 +24.313,E4 +24.313} C_DIS
 LIN_REL {X  -0.131,Y +67.751,A -1.956,E1 +0.039,E3 +32.889,E4 +32.889} C_DIS
 LIN_REL {X  +0.099,Y +84.776,A -0.269,E1 -0.006,E3 +42.702,E4 +42.702} C_DIS
 LIN_REL {X  +0.044,Y +130.298,A -0.006,E1 +0.010,E3 +65.859,E4 +65.859} C_DIS
 LIN_REL {X  +0.015,Y +82.894,A +0.000,E1 +0.002,E3 +41.923,E4 +41.923} C_DIS
 LIN_REL {X  +0.229,Y +64.686,A -0.000,E1 +0.028,E3 +32.885,E4 +32.885} C_DIS
 LIN_REL {X  +1.572,Y +50.485,A -0.000,E1 +0.179,E3 +26.750,E4 +26.750} C_DIS
 LIN_REL {X  +4.865,Y +37.753,A -0.000,E1 +0.538,E3 +22.734,E4 +22.734} C_DIS
 LIN_REL {X  +5.706,Y +18.991,A -0.003,E1 +0.650,E3 +13.649,E4 +13.649} C_DIS
 LIN_REL {X  +6.265,Y +12.499,A -0.022,E1 +0.756,E3 +10.406,E4 +10.406} C_DIS
 LIN_REL {X  +15.158,Y +19.045,A -1.102,E1 +2.023,E3 +17.751,E4 +17.751} C_DIS
 LIN_REL {X  +12.826,Y +10.517,A -6.112,E1 +2.407,E3 +11.809,E4 +11.809} C_DIS
 LIN_REL {X  +14.127,Y +9.091,A -4.080,E1 +3.025,E3 +14.920,E4 +14.920} C_DIS
 LIN_REL {X  +10.852,Y +6.631,A -11.421,E1 +4.753,E3 +15.223,E4 +15.223} C_DIS
 LIN_REL {X  +7.046,Y +5.188,A -5.925,E1 +3.770,E3 +13.435,E4 +13.435} C_DIS
 LIN_REL {X  +7.579,Y +10.826,A -0.245,E1 +3.228,E3 +24.777,E4 +24.777} C_DIS
 LIN_REL {X  +5.059,Y +16.661,A -1.045,E1 +3.916,E3 +39.392,E4 +39.392} C_DIS
 LIN_REL {X  +0.881,Y +17.128,A -0.045,E1 +9.223,E3 +63.826,E4 +63.826} C_DIS
 LIN_REL {X  -2.887,Y -0.939,A -0.000,E1 +9.258,E3 +44.429,E4 +44.429} C_DIS
 LIN_REL {X  -1.220,Y -6.635,A -0.000,E1 +5.253,E3 +20.403,E4 +20.403} C_DIS
 LIN_REL {X  -1.215,Y -20.716,A -0.000,E1 +13.844,E3 +29.271,E4 +29.271} C_DIS
 LIN_REL {X  -8.638,Y -16.150,A -0.000,E1 +12.315,E3 +27.428,E4 +27.428} C_DIS
 LIN_REL {X  -13.005,Y -10.723,A -0.000,E1 +17.718,E3 +21.350,E4 +21.350} C_DIS
 LIN_REL {X  -12.219,Y -8.304,A -0.000,E1 +12.922,E3 +14.158,E4 +14.158} C_DIS
 LIN_REL {X  -4.980,Y -2.322,A -0.000,E1 +2.443,E3 +9.173,E4 +9.173} C_DIS
 LIN_REL {X  -7.461,Y -6.696,A -0.000,E1 +6.664,E3 +9.513,E4 +9.513} C_DIS
 LIN_REL {X  -12.876,Y -13.291,A -0.000,E1 +8.881,E3 +8.328,E4 +8.328} C_DIS
 LIN_REL {X  -9.601,Y -11.045,A -0.000,E1 +6.285,E3 +17.742,E4 +17.742} C_DIS
ENDFOR

HALT
LIN {X -173.020,Y 1394.835,Z 0.000,A -30.000, B 0.00, C 0.00,E1 60.710}
HALT

; PLY 35 OF 41 (Connector)

; ANGLE 51.0 (Not valid for Circ layers and non-tubes)
$APO.CDIS=85
$VEL_EXTAX[1]=100
FOR N_CYC=1 to 1
 LIN_REL {X  +0.000,Y -14.724,A +0.000,E1 +1.729,E3 +9.078,E4 +9.078} C_DIS
 LIN_REL {X  +0.000,Y -6.122,A +0.000,E1 +1.066,E3 +8.147,E4 +8.147} C_DIS
 LIN_REL {X  +0.000,Y +1.925,A +0.000,E1 +0.860,E3 +2.808,E4 +2.808} C_DIS
 LIN_REL {X  +0.000,Y -32.386,A +0.000,E1 +4.362,E3 +9.711,E4 +9.711} C_DIS
 LIN_REL {X  +0.000,Y -44.374,A +0.002,E1 +1.937,E3 +16.647,E4 +16.647} C_DIS
 LIN_REL {X  +0.000,Y -21.393,A +1.102,E1 -0.147,E3 +9.500,E4 +9.500} C_DIS
 LIN_REL {X  +0.000,Y -10.548,A +0.301,E1 +0.334,E3 +7.027,E4 +7.027} C_DIS
 LIN_REL {X  +0.000,Y -31.525,A +7.745,E1 -0.447,E3 +14.529,E4 +14.529} C_DIS
 LIN_REL {X  +0.000,Y -38.278,A +9.573,E1 -1.050,E3 +18.794,E4 +18.794} C_DIS
 LIN_REL {X  +0.000,Y -32.357,A +3.190,E1 +0.107,E3 +18.386,E4 +18.386} C_DIS
 LIN_REL {X  +0.000,Y -46.374,A +5.461,E1 -1.367,E3 +30.774,E4 +30.774} C_DIS
 LIN_REL {X  +0.000,Y -53.318,A +2.455,E1 -2.739,E3 +50.842,E4 +50.842} C_DIS
 LIN_REL {X  +0.000,Y -59.888,A +0.166,E1 -3.923,E3 +69.122,E4 +69.122} C_DIS
 LIN_REL {X  +0.000,Y -66.146,A +0.005,E1 -4.415,E3 +84.729,E4 +84.729} C_DIS
 LIN_REL {X  +0.000,Y -65.741,A -0.000,E1 -4.684,E3 +95.805,E4 +95.805} C_DIS
 LIN_REL {X  +0.000,Y -60.683,A +0.000,E1 -4.791,E3 +102.469,E4 +102.469} C_DIS
 LIN_REL {X  +0.000,Y -45.559,A +0.000,E1 -4.045,E3 +89.055,E4 +89.055} C_DIS
 LIN_REL {X  +0.000,Y -34.164,A +0.000,E1 -3.413,E3 +76.242,E4 +76.242} C_DIS
 LIN_REL {X  +0.000,Y -24.251,A +0.001,E1 -3.015,E3 +60.834,E4 +60.834} C_DIS
 LIN_REL {X  +0.000,Y -12.884,A +0.001,E1 -2.636,E3 +35.043,E4 +35.043} C_DIS
 LIN_REL {X  +0.000,Y -8.288,A +0.003,E1 -1.656,E3 +23.851,E4 +23.851} C_DIS
 LIN_REL {X  +0.000,Y -13.152,A +0.006,E1 -0.795,E3 +38.808,E4 +38.808} C_DIS
 LIN_REL {X  +0.000,Y -18.137,A +0.022,E1 -2.704,E3 +60.125,E4 +60.125} C_DIS
 LIN_REL {X  +0.000,Y -20.170,A +0.072,E1 -3.685,E3 +78.480,E4 +78.480} C_DIS
 LIN_REL {X  +0.000,Y -19.522,A +0.221,E1 -4.650,E3 +94.926,E4 +94.926} C_DIS
 LIN_REL {X  +0.000,Y -12.880,A +0.450,E1 -4.647,E3 +86.087,E4 +86.087} C_DIS
 LIN_REL {X  +0.000,Y -6.280,A +0.610,E1 -4.221,E3 +64.073,E4 +64.073} C_DIS
 LIN_REL {X  +0.000,Y -2.966,A +1.172,E1 -6.561,E3 +81.118,E4 +81.118} C_DIS
 LIN_REL {X  +0.000,Y +1.168,A +1.294,E1 -6.149,E3 +84.685,E4 +84.685} C_DIS
 LIN_REL {X  +0.000,Y +1.625,A +0.536,E1 -1.999,E3 +32.839,E4 +32.839} C_DIS
 LIN_REL {X  +0.000,Y +2.557,A +0.507,E1 -1.514,E3 +28.039,E4 +28.039} C_DIS
ENDFOR

HALT
LIN {X -173.020,Y 600.000,Z 0.000,A 0.000, B 0.00, C 0.00,E1 -0.000}
HALT

; PLY 36 OF 41 (Circ)

; ANGLE 51.0 (Not valid for Circ layers and non-tubes)
$APO.CDIS=85
$VEL_EXTAX[1]=100
FOR N_CYC=1 to 1
 LIN_REL {X  +0.000,Y +0.000,A +0.000,E1 +0.000,E3 +13.889,E4 +13.889} C_DIS
 LIN_REL {X  +0.000,Y +6.750,A +0.000,E1 -0.925,E3 +500.000,E4 +500.000} C_DIS
 LIN_REL {X  +0.000,Y +706.500,A +0.000,E1 -0.000,E3 +52333.333,E4 +52333.333} C_DIS
 LIN_REL {X  +0.000,Y +6.750,A +0.000,E1 +0.925,E3 +500.000,E4 +500.000} C_DIS
 LIN_REL {X  +0.000,Y +0.000,A +0.000,E1 +0.000,E3 +500.000,E4 +500.000} C_DIS
 LIN_REL {X  +0.000,Y -6.750,A +0.000,E1 +0.925,E3 +500.000,E4 +500.000} C_DIS
 LIN_REL {X  +0.000,Y -706.500,A +0.000,E1 +0.000,E3 +52333.334,E4 +52333.334} C_DIS
 LIN_REL {X  +0.000,Y -6.750,A +0.000,E1 -0.925,E3 +500.000,E4 +500.000} C_DIS
 LIN_REL {X  +0.000,Y +0.000,A +0.000,E1 +0.000,E3 +13.889,E4 +13.889} C_DIS
ENDFOR

HALT
LIN {X -172.689,Y 614.180,Z 0.000,A 2.576, B 0.00, C 0.00,E1 -4.273}
HALT

; PLY 37 OF 41 (Helical)

; ANGLE 51.0 (Not valid for Circ layers and non-tubes)
$APO.CDIS=85
$VEL_EXTAX[1]=100
FOR N_CYC=1 to 7
 LIN_REL {X  +1.465,Y +3.444,A -0.525,E1 -0.825,E3 +54.356,E4 +54.356} C_DIS
 LIN_REL {X  +1.270,Y +4.602,A -0.549,E1 -1.004,E3 +70.370,E4 +70.370} C_DIS
 LIN_REL {X  -0.330,Y +9.503,A -0.420,E1 -1.842,E3 +93.539,E4 +93.539} C_DIS
 LIN_REL {X  +0.202,Y +11.237,A -0.395,E1 -0.667,E3 +114.359,E4 +114.359} C_DIS
 LIN_REL {X  +0.023,Y +12.008,A -0.186,E1 +0.142,E3 +136.039,E4 +136.039} C_DIS
 LIN_REL {X  -0.178,Y +14.891,A -0.255,E1 +0.225,E3 +167.797,E4 +167.797} C_DIS
 LIN_REL {X  +0.174,Y +10.952,A -0.115,E1 +0.080,E3 +123.259,E4 +123.259} C_DIS
 LIN_REL {X  +0.101,Y +13.667,A -0.049,E1 +0.039,E3 +155.961,E4 +155.961} C_DIS
 LIN_REL {X  -0.129,Y +10.786,A -0.024,E1 +0.032,E3 +121.944,E4 +121.944} C_DIS
 LIN_REL {X  -0.050,Y +13.320,A -0.033,E1 +0.027,E3 +150.010,E4 +150.010} C_DIS
 LIN_REL {X  +0.087,Y +10.657,A -0.010,E1 +0.003,E3 +120.708,E4 +120.708} C_DIS
 LIN_REL {X  +0.075,Y +13.623,A -0.007,E1 +0.000,E3 +154.041,E4 +154.041} C_DIS
 LIN_REL {X  +0.050,Y +14.697,A -0.004,E1 +0.000,E3 +166.189,E4 +166.189} C_DIS
 LIN_REL {X  +0.025,Y +417.295,A -0.007,E1 +0.005,E3 +4719.370,E4 +4719.370} C_DIS
 LIN_REL {X  -0.025,Y +10.953,A -0.003,E1 +0.004,E3 +123.948,E4 +123.948} C_DIS
 LIN_REL {X  -0.036,Y +10.902,A -0.004,E1 +0.007,E3 +123.423,E4 +123.423} C_DIS
 LIN_REL {X  -0.057,Y +12.241,A -0.007,E1 +0.011,E3 +138.570,E4 +138.570} C_DIS
 LIN_REL {X  -0.084,Y +12.573,A -0.012,E1 +0.017,E3 +142.338,E4 +142.338} C_DIS
 LIN_REL {X  +0.030,Y +15.208,A -0.032,E1 +0.023,E3 +170.981,E4 +170.981} C_DIS
 LIN_REL {X  +0.151,Y +11.173,A -0.034,E1 +0.017,E3 +126.855,E4 +126.855} C_DIS
 LIN_REL {X  -0.027,Y +11.858,A -0.033,E1 +0.039,E3 +134.900,E4 +134.900} C_DIS
 LIN_REL {X  -0.241,Y +11.037,A -0.074,E1 +0.084,E3 +124.579,E4 +124.579} C_DIS
 LIN_REL {X  +0.071,Y +10.699,A -0.170,E1 +0.138,E3 +120.993,E4 +120.993} C_DIS
 LIN_REL {X  +0.333,Y +10.994,A -0.216,E1 +0.170,E3 +124.398,E4 +124.398} C_DIS
 LIN_REL {X  -0.055,Y +10.357,A -0.184,E1 +0.248,E3 +119.276,E4 +119.276} C_DIS
 LIN_REL {X  +0.344,Y +7.121,A -0.419,E1 +1.546,E3 +106.263,E4 +106.263} C_DIS
 LIN_REL {X  +0.387,Y +2.369,A -0.336,E1 +3.294,E3 +111.540,E4 +111.540} C_DIS
 LIN_REL {X  +0.032,Y -0.422,A -0.090,E1 +4.038,E3 +233.310,E4 +233.310} C_DIS
 LIN_REL {X  -0.384,Y -11.095,A +0.152,E1 +3.781,E3 +238.876,E4 +238.876} C_DIS
 LIN_REL {X  -0.489,Y -10.316,A +0.398,E1 +2.165,E3 +122.288,E4 +122.288} C_DIS
 LIN_REL {X  -0.138,Y -11.066,A +0.391,E1 +0.931,E3 +111.158,E4 +111.158} C_DIS
 LIN_REL {X  +0.077,Y -11.239,A +0.185,E1 +0.011,E3 +124.940,E4 +124.940} C_DIS
 LIN_REL {X  -0.248,Y -10.922,A +0.174,E1 -0.167,E3 +123.950,E4 +123.950} C_DIS
 LIN_REL {X  +0.052,Y -10.742,A +0.143,E1 -0.110,E3 +120.969,E4 +120.969} C_DIS
 LIN_REL {X  +0.254,Y -11.583,A +0.072,E1 -0.041,E3 +130.472,E4 +130.472} C_DIS
 LIN_REL {X  -0.031,Y -11.365,A +0.027,E1 -0.030,E3 +129.850,E4 +129.850} C_DIS
 LIN_REL {X  -0.159,Y -15.752,A +0.038,E1 -0.042,E3 +177.684,E4 +177.684} C_DIS
 LIN_REL {X  +0.053,Y -12.009,A +0.016,E1 -0.009,E3 +135.406,E4 +135.406} C_DIS
 LIN_REL {X  +0.095,Y -14.965,A +0.010,E1 -0.002,E3 +169.306,E4 +169.306} C_DIS
 LIN_REL {X  +0.050,Y -12.293,A +0.005,E1 -0.000,E3 +139.010,E4 +139.010} C_DIS
 LIN_REL {X  +0.044,Y -423.519,A +0.009,E1 -0.006,E3 +4789.215,E4 +4789.215} C_DIS
 LIN_REL {X  -0.025,Y -10.955,A +0.002,E1 -0.003,E3 +123.948,E4 +123.948} C_DIS
 LIN_REL {X  -0.036,Y -10.903,A +0.004,E1 -0.007,E3 +123.422,E4 +123.422} C_DIS
 LIN_REL {X  -0.057,Y -12.243,A +0.007,E1 -0.010,E3 +138.570,E4 +138.570} C_DIS
 LIN_REL {X  -0.085,Y -12.575,A +0.011,E1 -0.017,E3 +142.339,E4 +142.339} C_DIS
 LIN_REL {X  +0.031,Y -15.210,A +0.035,E1 -0.026,E3 +170.983,E4 +170.983} C_DIS
 LIN_REL {X  +0.153,Y -11.176,A +0.038,E1 -0.021,E3 +126.861,E4 +126.861} C_DIS
 LIN_REL {X  -0.024,Y -11.861,A +0.039,E1 -0.043,E3 +134.911,E4 +134.911} C_DIS
 LIN_REL {X  -0.237,Y -11.039,A +0.086,E1 -0.094,E3 +124.596,E4 +124.596} C_DIS
 LIN_REL {X  +0.079,Y -10.702,A +0.196,E1 -0.161,E3 +121.016,E4 +121.016} C_DIS
 LIN_REL {X  +0.349,Y -10.996,A +0.246,E1 -0.195,E3 +124.429,E4 +124.429} C_DIS
 LIN_REL {X  -0.072,Y -10.328,A +0.200,E1 -0.272,E3 +119.244,E4 +119.244} C_DIS
 LIN_REL {X  +0.057,Y -6.858,A +0.483,E1 -1.842,E3 +108.153,E4 +108.153} C_DIS
 LIN_REL {X  +0.297,Y -1.997,A +0.542,E1 -3.060,E3 +94.519,E4 +94.519} C_DIS
 LIN_REL {X  -1.625,Y +2.728,A +0.407,E1 -3.525,E3 +74.363,E4 +74.363} C_DIS
 LIN_REL {X  -1.589,Y +3.236,A +0.277,E1 -3.056,E3 +81.635,E4 +81.635} C_DIS
ENDFOR

HALT
LIN {X -173.745,Y 605.092,Z 0.000,A -0.243, B 0.00, C 0.00,E1 3.924}
HALT

; PLY 38 OF 41 (Connector)

; ANGLE 51.0 (Not valid for Circ layers and non-tubes)
$APO.CDIS=85
$VEL_EXTAX[1]=100
FOR N_CYC=1 to 1
 LIN_REL {X  +0.000,Y -2.053,A +1.455,E1 -0.802,E3 +36.620,E4 +36.620} C_DIS
 LIN_REL {X  +0.000,Y -2.632,A +1.886,E1 -1.057,E3 +47.616,E4 +47.616} C_DIS
 LIN_REL {X  +0.000,Y -2.033,A +4.472,E1 -4.724,E3 +58.372,E4 +58.372} C_DIS
 LIN_REL {X  +0.000,Y -1.567,A +4.526,E1 -5.026,E3 +50.949,E4 +50.949} C_DIS
 LIN_REL {X  +0.000,Y +0.840,A +2.771,E1 -3.134,E3 +27.244,E4 +27.244} C_DIS
 LIN_REL {X  +0.000,Y +2.353,A +3.734,E1 -4.265,E3 +33.735,E4 +33.735} C_DIS
ENDFOR

HALT
LIN {X -173.929,Y 600.000,Z 0.000,A 0.000, B 0.00, C 0.00,E1 -0.000}
HALT

; PLY 39 OF 41 (Circ)

; ANGLE 51.0 (Not valid for Circ layers and non-tubes)
$APO.CDIS=85
$VEL_EXTAX[1]=100
FOR N_CYC=1 to 1
 LIN_REL {X  +0.000,Y +0.000,A +0.000,E1 +0.000,E3 +13.889,E4 +13.889} C_DIS
 LIN_REL {X  +0.000,Y +6.750,A +0.000,E1 -0.919,E3 +500.000,E4 +500.000} C_DIS
 LIN_REL {X  +0.000,Y +706.500,A +0.000,E1 -0.000,E3 +52333.333,E4 +52333.333} C_DIS
 LIN_REL {X  +0.000,Y +6.750,A +0.000,E1 +0.919,E3 +500.000,E4 +500.000} C_DIS
 LIN_REL {X  +0.000,Y +0.000,A +0.000,E1 +0.000,E3 +500.000,E4 +500.000} C_DIS
 LIN_REL {X  +0.000,Y -6.750,A +0.000,E1 +0.919,E3 +500.000,E4 +500.000} C_DIS
 LIN_REL {X  +0.000,Y -706.500,A +0.000,E1 +0.000,E3 +52333.334,E4 +52333.334} C_DIS
 LIN_REL {X  +0.000,Y -6.750,A +0.000,E1 -0.919,E3 +500.000,E4 +500.000} C_DIS
 LIN_REL {X  +0.000,Y +0.000,A +0.000,E1 +0.000,E3 +13.889,E4 +13.889} C_DIS
ENDFOR

HALT
LIN {X -174.367,Y 600.000,Z 0.000,A 20.868, B 0.00, C 0.00,E1 -16.820}
HALT

; PLY 40 OF 41 (Connector)

; ANGLE 51.0 (Not valid for Circ layers and non-tubes)
$APO.CDIS=85
$VEL_EXTAX[1]=100
FOR N_CYC=1 to 1
 LIN_REL {X  +0.000,Y +4.559,A -2.378,E1 -1.708,E3 +17.035,E4 +17.035} C_DIS
 LIN_REL {X  +0.000,Y +8.901,A -9.179,E1 +1.843,E3 +33.219,E4 +33.219} C_DIS
 LIN_REL {X  +0.000,Y +10.537,A -7.819,E1 +3.015,E3 +43.632,E4 +43.632} C_DIS
 LIN_REL {X  +0.000,Y +7.331,A -1.966,E1 -0.006,E3 +30.751,E4 +30.751} C_DIS
 LIN_REL {X  +0.000,Y +12.535,A +0.300,E1 -2.469,E3 +50.163,E4 +50.163} C_DIS
 LIN_REL {X  +0.000,Y +19.044,A +0.699,E1 -3.807,E3 +68.517,E4 +68.517} C_DIS
 LIN_REL {X  +0.000,Y +28.474,A -0.256,E1 -3.915,E3 +85.775,E4 +85.775} C_DIS
 LIN_REL {X  +0.000,Y +31.574,A -0.171,E1 -3.644,E3 +81.335,E4 +81.335} C_DIS
 LIN_REL {X  +0.000,Y +27.872,A -0.059,E1 -2.843,E3 +63.333,E4 +63.333} C_DIS
 LIN_REL {X  +0.000,Y +21.882,A -0.021,E1 -2.103,E3 +44.434,E4 +44.434} C_DIS
 LIN_REL {X  +0.000,Y +15.657,A -0.007,E1 -1.476,E3 +26.959,E4 +26.959} C_DIS
 LIN_REL {X  +0.000,Y +15.587,A -0.005,E1 -1.217,E3 +32.587,E4 +32.587} C_DIS
 LIN_REL {X  +0.000,Y +15.565,A -0.003,E1 -0.845,E3 +27.491,E4 +27.491} C_DIS
 LIN_REL {X  +0.000,Y +25.850,A -0.002,E1 -1.844,E3 +43.382,E4 +43.382} C_DIS
 LIN_REL {X  +0.000,Y +37.398,A -0.001,E1 -2.665,E3 +58.012,E4 +58.012} C_DIS
 LIN_REL {X  +0.000,Y +49.562,A -0.000,E1 -3.227,E3 +69.344,E4 +69.344} C_DIS
 LIN_REL {X  +0.000,Y +66.029,A -0.000,E1 -3.841,E3 +81.459,E4 +81.459} C_DIS
 LIN_REL {X  +0.000,Y +74.064,A -0.000,E1 -3.823,E3 +79.394,E4 +79.394} C_DIS
 LIN_REL {X  +0.000,Y +78.480,A -0.000,E1 -3.613,E3 +72.797,E4 +72.797} C_DIS
 LIN_REL {X  +0.000,Y +83.444,A -0.000,E1 -3.445,E3 +66.738,E4 +66.738} C_DIS
 LIN_REL {X  +0.000,Y +85.196,A -0.006,E1 -3.169,E3 +58.488,E4 +58.488} C_DIS
 LIN_REL {X  +0.000,Y +70.867,A -0.047,E1 -2.395,E3 +42.252,E4 +42.252} C_DIS
 LIN_REL {X  +0.000,Y +58.885,A -0.207,E1 -1.802,E3 +31.372,E4 +31.372} C_DIS
 LIN_REL {X  +0.000,Y +42.166,A +0.158,E1 -1.226,E3 +20.776,E4 +20.776} C_DIS
 LIN_REL {X  +0.000,Y +28.889,A +0.140,E1 -1.843,E3 +17.210,E4 +17.210} C_DIS
 LIN_REL {X  +0.000,Y +27.977,A -7.459,E1 +0.890,E3 +22.254,E4 +22.254} C_DIS
 LIN_REL {X  +0.000,Y +27.613,A -13.515,E1 +6.413,E3 +25.344,E4 +25.344} C_DIS
 LIN_REL {X  +0.000,Y +15.120,A -6.445,E1 +5.375,E3 +14.706,E4 +14.706} C_DIS
 LIN_REL {X  +0.000,Y +8.967,A +1.301,E1 +1.175,E3 +8.226,E4 +8.226} C_DIS
 LIN_REL {X  +0.000,Y +3.091,A +7.203,E1 -7.145,E3 +1.490,E4 +1.490} C_DIS
 LIN_REL {X  +0.000,Y +0.977,A +3.135,E1 -2.864,E3 +1.198,E4 +1.198} C_DIS
 LIN_REL {X  +0.000,Y +8.005,A -3.541,E1 +1.150,E3 +4.491,E4 +4.491} C_DIS
 LIN_REL {X  +0.000,Y +11.954,A -8.088,E1 +4.430,E3 +21.642,E4 +21.642} C_DIS
 LIN_REL {X  +0.000,Y +7.284,A -2.604,E1 +5.230,E3 +32.617,E4 +32.617} C_DIS
 LIN_REL {X  +0.000,Y -5.042,A -0.025,E1 +5.087,E3 +29.898,E4 +29.898} C_DIS
 LIN_REL {X  +0.000,Y -9.995,A -0.000,E1 +3.784,E3 +23.405,E4 +23.405} C_DIS
 LIN_REL {X  +0.000,Y -1.454,A -0.000,E1 -3.443,E3 +7.160,E4 +7.160} C_DIS
 LIN_REL {X  +0.000,Y -22.869,A -0.000,E1 +9.715,E3 +21.163,E4 +21.163} C_DIS
 LIN_REL {X  +0.000,Y -32.953,A -0.000,E1 +14.427,E3 +23.904,E4 +23.904} C_DIS
 LIN_REL {X  +0.000,Y -26.834,A -0.000,E1 +8.677,E3 +15.257,E4 +15.257} C_DIS
 LIN_REL {X  +0.000,Y -19.451,A -0.000,E1 +13.726,E3 +9.382,E4 +9.382} C_DIS
 LIN_REL {X  +0.000,Y -15.096,A -0.000,E1 +9.367,E3 +6.878,E4 +6.878} C_DIS
 LIN_REL {X  +0.000,Y -18.052,A -0.000,E1 +6.734,E3 +8.146,E4 +8.146} C_DIS
 LIN_REL {X  +0.000,Y -24.618,A -0.000,E1 +16.402,E3 +9.116,E4 +9.116} C_DIS
 LIN_REL {X  +0.000,Y -26.056,A -0.000,E1 +14.649,E3 +7.865,E4 +7.865} C_DIS
 LIN_REL {X  +0.000,Y -18.514,A -0.000,E1 +5.040,E3 +6.844,E4 +6.844} C_DIS
 LIN_REL {X  +0.000,Y -8.039,A -0.000,E1 +2.077,E3 +4.661,E4 +4.661} C_DIS
 LIN_REL {X  +0.000,Y -6.143,A -0.000,E1 +1.727,E3 +3.270,E4 +3.270} C_DIS
 LIN_REL {X  +0.000,Y -5.546,A -0.000,E1 +1.562,E3 +1.904,E4 +1.904} C_DIS
 LIN_REL {X  +0.000,Y -20.005,A -0.000,E1 +6.111,E3 +4.593,E4 +4.593} C_DIS
 LIN_REL {X  +0.000,Y -39.055,A -0.000,E1 +6.285,E3 +10.547,E4 +10.547} C_DIS
 LIN_REL {X  +0.000,Y -38.295,A +0.012,E1 +2.561,E3 +13.005,E4 +13.005} C_DIS
 LIN_REL {X  +0.000,Y -16.943,A +1.263,E1 +0.119,E3 +6.489,E4 +6.489} C_DIS
 LIN_REL {X  +0.000,Y -8.457,A -0.549,E1 +1.069,E3 +4.499,E4 +4.499} C_DIS
 LIN_REL {X  +0.000,Y -30.840,A +6.220,E1 -0.029,E3 +11.848,E4 +11.848} C_DIS
 LIN_REL {X  +0.000,Y -37.631,A +8.258,E1 -0.589,E3 +14.992,E4 +14.992} C_DIS
 LIN_REL {X  +0.000,Y -22.458,A +4.377,E1 -0.154,E3 +8.996,E4 +8.996} C_DIS
 LIN_REL {X  +0.000,Y -10.276,A +0.668,E1 +0.780,E3 +4.140,E4 +4.140} C_DIS
 LIN_REL {X  +0.000,Y +0.300,A -5.457,E1 +2.637,E3 +2.104,E4 +2.104} C_DIS
 LIN_REL {X  +0.000,Y -20.823,A +0.351,E1 -0.947,E3 +8.674,E4 +8.674} C_DIS
 LIN_REL {X  +0.000,Y -35.345,A +6.934,E1 -1.454,E3 +15.241,E4 +15.241} C_DIS
 LIN_REL {X  +0.000,Y -44.162,A +7.346,E1 -1.058,E3 +19.173,E4 +19.173} C_DIS
 LIN_REL {X  +0.000,Y -30.483,A +0.860,E1 +1.249,E3 +12.889,E4 +12.889} C_DIS
 LIN_REL {X  +0.000,Y -43.565,A -0.492,E1 +0.089,E3 +20.759,E4 +20.759} C_DIS
 LIN_REL {X  +0.000,Y -58.236,A +0.184,E1 -0.028,E3 +28.964,E4 +28.964} C_DIS
 LIN_REL {X  +0.000,Y -438.643,A +0.028,E1 -0.006,E3 +218.279,E4 +218.279} C_DIS
 LIN_REL {X  +0.000,Y -53.488,A +0.028,E1 -0.008,E3 +26.634,E4 +26.634} C_DIS
 LIN_REL {X  +0.000,Y -38.328,A +0.115,E1 -0.021,E3 +19.149,E4 +19.149} C_DIS
 LIN_REL {X  +0.000,Y -23.907,A +0.209,E1 -0.081,E3 +12.057,E4 +12.057} C_DIS
 LIN_REL {X  +0.000,Y -10.659,A +0.093,E1 -0.011,E3 +5.524,E4 +5.524} C_DIS
 LIN_REL {X  +0.000,Y -26.389,A -0.592,E1 +1.171,E3 +15.808,E4 +15.808} C_DIS
 LIN_REL {X  +0.000,Y -32.929,A +0.527,E1 +0.884,E3 +23.184,E4 +23.184} C_DIS
 LIN_REL {X  +0.000,Y -28.724,A +5.738,E1 -3.340,E3 +21.987,E4 +21.987} C_DIS
 LIN_REL {X  +0.000,Y -19.323,A +11.056,E1 -6.172,E3 +14.816,E4 +14.816} C_DIS
 LIN_REL {X  +0.000,Y -10.675,A +6.580,E1 -2.085,E3 +7.429,E4 +7.429} C_DIS
 LIN_REL {X  +0.000,Y -7.681,A -2.020,E1 +4.709,E3 +2.086,E4 +2.086} C_DIS
 LIN_REL {X  +0.000,Y -6.687,A -5.578,E1 +2.865,E3 +3.149,E4 +3.149} C_DIS
 LIN_REL {X  +0.000,Y -9.810,A +4.032,E1 -0.670,E3 +15.441,E4 +15.441} C_DIS
 LIN_REL {X  +0.000,Y -7.464,A +6.631,E1 -3.320,E3 +19.334,E4 +19.334} C_DIS
 LIN_REL {X  +0.000,Y -1.199,A +3.148,E1 -5.009,E3 +36.488,E4 +36.488} C_DIS
 LIN_REL {X  +0.000,Y +16.477,A +0.030,E1 -5.641,E3 +39.056,E4 +39.056} C_DIS
 LIN_REL {X  +0.000,Y +17.291,A -0.000,E1 -3.889,E3 +19.769,E4 +19.769} C_DIS
 LIN_REL {X  +0.000,Y -0.629,A -0.000,E1 +3.998,E3 +4.642,E4 +4.642} C_DIS
 LIN_REL {X  +0.000,Y +7.600,A -0.000,E1 +0.503,E3 +5.679,E4 +5.679} C_DIS
 LIN_REL {X  +0.000,Y +27.592,A -0.000,E1 -8.333,E3 +16.682,E4 +16.682} C_DIS
 LIN_REL {X  +0.000,Y +39.453,A -0.000,E1 -13.131,E3 +20.482,E4 +20.482} C_DIS
 LIN_REL {X  +0.000,Y +15.804,A -0.000,E1 -5.032,E3 +7.140,E4 +7.140} C_DIS
 LIN_REL {X  +0.000,Y +22.657,A -0.000,E1 -3.719,E3 +9.016,E4 +9.016} C_DIS
 LIN_REL {X  +0.000,Y +20.340,A -0.000,E1 -13.430,E3 +7.298,E4 +7.298} C_DIS
 LIN_REL {X  +0.000,Y +15.446,A -0.000,E1 -11.506,E3 +5.256,E4 +5.256} C_DIS
 LIN_REL {X  +0.000,Y +11.276,A -0.000,E1 -3.636,E3 +3.652,E4 +3.652} C_DIS
 LIN_REL {X  +0.000,Y +13.901,A -0.000,E1 -4.625,E3 +4.418,E4 +4.418} C_DIS
 LIN_REL {X  +0.000,Y +18.769,A -0.000,E1 -13.809,E3 +5.509,E4 +5.509} C_DIS
 LIN_REL {X  +0.000,Y +26.656,A -0.000,E1 -18.408,E3 +6.807,E4 +6.807} C_DIS
 LIN_REL {X  +0.000,Y +13.181,A -0.000,E1 -7.268,E3 +2.888,E4 +2.888} C_DIS
 LIN_REL {X  +0.000,Y +3.121,A -0.000,E1 -0.844,E3 +1.203,E4 +1.203} C_DIS
 LIN_REL {X  +0.000,Y -11.887,A -0.000,E1 +5.039,E3 +0.710,E4 +0.710} C_DIS
 LIN_REL {X  +0.000,Y -0.568,A -0.000,E1 -0.573,E3 +0.473,E4 +0.473} C_DIS
 LIN_REL {X  +0.000,Y +24.961,A -0.000,E1 -10.204,E3 +13.362,E4 +13.362} C_DIS
ENDFOR

HALT
LIN {X -153.872,Y 525.962,Z 0.000,A 30.000, B 0.00, C 0.00,E1 -57.784}
HALT

; PLY 41 OF 41 (Helical)

; ANGLE 51.0 (Not valid for Circ layers and non-tubes)
$APO.CDIS=85
$VEL_EXTAX[1]=100
FOR N_CYC=1 to 58
 LIN_REL {X  -7.305,Y +14.468,A +0.000,E1 -4.453,E3 +12.303,E4 +12.303} C_DIS
 LIN_REL {X  -5.453,Y +18.676,A +0.000,E1 -4.421,E3 +7.585,E4 +7.585} C_DIS
 LIN_REL {X  -6.082,Y +36.611,A +0.000,E1 -4.437,E3 +11.713,E4 +11.713} C_DIS
 LIN_REL {X  -1.232,Y +28.952,A -0.256,E1 -1.178,E3 +9.815,E4 +9.815} C_DIS
 LIN_REL {X  -0.203,Y +18.662,A -1.813,E1 -0.206,E3 +6.647,E4 +6.647} C_DIS
 LIN_REL {X  +0.127,Y +17.917,A -0.233,E1 -0.636,E3 +6.698,E4 +6.698} C_DIS
 LIN_REL {X  +0.275,Y +25.734,A -9.279,E1 +0.239,E3 +9.938,E4 +9.938} C_DIS
 LIN_REL {X  +0.048,Y +34.019,A -8.736,E1 +0.741,E3 +13.493,E4 +13.493} C_DIS
 LIN_REL {X  -0.315,Y +30.547,A -1.590,E1 +0.152,E3 +12.432,E4 +12.432} C_DIS
 LIN_REL {X  +0.053,Y +24.256,A +2.116,E1 -0.838,E3 +10.170,E4 +10.170} C_DIS
 LIN_REL {X  +0.403,Y +17.214,A +2.718,E1 -0.460,E3 +7.396,E4 +7.396} C_DIS
 LIN_REL {X  +0.388,Y +19.399,A -6.229,E1 +0.394,E3 +8.483,E4 +8.483} C_DIS
 LIN_REL {X  +0.224,Y +27.009,A -6.583,E1 +0.862,E3 +12.061,E4 +12.061} C_DIS
 LIN_REL {X  -0.248,Y +33.773,A +0.050,E1 +0.237,E3 +15.496,E4 +15.496} C_DIS
 LIN_REL {X  -0.587,Y +47.736,A +0.105,E1 -0.375,E3 +22.826,E4 +22.826} C_DIS
 LIN_REL {X  +0.050,Y +65.806,A -0.252,E1 -0.021,E3 +32.529,E4 +32.529} C_DIS
 LIN_REL {X  +0.059,Y +78.835,A -0.018,E1 +0.011,E3 +39.144,E4 +39.144} C_DIS
 LIN_REL {X  +0.010,Y +89.987,A +0.000,E1 +0.003,E3 +44.710,E4 +44.710} C_DIS
 LIN_REL {X  +0.046,Y +82.730,A -0.000,E1 +0.005,E3 +41.141,E4 +41.141} C_DIS
 LIN_REL {X  +0.883,Y +69.511,A -0.000,E1 +0.105,E3 +35.221,E4 +35.221} C_DIS
 LIN_REL {X  +6.641,Y +54.294,A -0.001,E1 +0.723,E3 +31.863,E4 +31.863} C_DIS
 LIN_REL {X  +13.532,Y +35.009,A -0.052,E1 +1.596,E3 +26.229,E4 +26.229} C_DIS
 LIN_REL {X  +11.420,Y +15.097,A -0.116,E1 +1.342,E3 +13.380,E4 +13.380} C_DIS
 LIN_REL {X  +8.333,Y +7.717,A -4.116,E1 +1.726,E3 +7.952,E4 +7.952} C_DIS
 LIN_REL {X  +8.029,Y +6.640,A -6.460,E1 +2.007,E3 +7.989,E4 +7.989} C_DIS
 LIN_REL {X  +6.575,Y +4.585,A +1.580,E1 +0.616,E3 +6.841,E4 +6.841} C_DIS
 LIN_REL {X  +9.734,Y +5.961,A -5.460,E1 +2.811,E3 +11.447,E4 +11.447} C_DIS
 LIN_REL {X  +9.924,Y +6.216,A -10.473,E1 +4.699,E3 +15.116,E4 +15.116} C_DIS
 LIN_REL {X  +8.239,Y +7.385,A -4.703,E1 +4.106,E3 +18.706,E4 +18.706} C_DIS
 LIN_REL {X  +8.190,Y +17.902,A -0.199,E1 +4.751,E3 +42.042,E4 +42.042} C_DIS
 LIN_REL {X  +2.362,Y +18.629,A +0.000,E1 +7.264,E3 +58.002,E4 +58.002} C_DIS
 LIN_REL {X  -2.342,Y +3.927,A +0.000,E1 +8.910,E3 +47.993,E4 +47.993} C_DIS
 LIN_REL {X  -1.741,Y -8.116,A +0.000,E1 +8.093,E3 +31.764,E4 +31.764} C_DIS
 LIN_REL {X  -1.699,Y -22.944,A +0.000,E1 +15.398,E3 +34.494,E4 +34.494} C_DIS
 LIN_REL {X  -10.315,Y -14.340,A +0.000,E1 +15.459,E3 +29.387,E4 +29.387} C_DIS
 LIN_REL {X  -12.647,Y -8.839,A +0.000,E1 +16.104,E3 +19.831,E4 +19.831} C_DIS
 LIN_REL {X  -8.491,Y -5.195,A +0.000,E1 +7.614,E3 +10.135,E4 +10.135} C_DIS
 LIN_REL {X  -11.440,Y -9.015,A +0.000,E1 +8.162,E3 +16.997,E4 +16.997} C_DIS
 LIN_REL {X  -17.593,Y -18.930,A +0.000,E1 +14.217,E3 +22.332,E4 +22.332} C_DIS
 LIN_REL {X  -11.791,Y -17.632,A +0.000,E1 +7.196,E3 +14.766,E4 +14.766} C_DIS
 LIN_REL {X  -7.110,Y -18.114,A +0.000,E1 +4.466,E3 +9.832,E4 +9.832} C_DIS
 LIN_REL {X  -7.164,Y -35.378,A +0.000,E1 +5.319,E3 +11.317,E4 +11.317} C_DIS
 LIN_REL {X  -1.872,Y -33.568,A +0.079,E1 +1.757,E3 +11.234,E4 +11.234} C_DIS
 LIN_REL {X  -0.210,Y -19.167,A +2.371,E1 +0.088,E3 +6.787,E4 +6.787} C_DIS
 LIN_REL {X  +0.063,Y -15.697,A -1.189,E1 +0.652,E3 +5.800,E4 +5.800} C_DIS
 LIN_REL {X  +0.221,Y -21.329,A +7.311,E1 -0.034,E3 +8.151,E4 +8.151} C_DIS
 LIN_REL {X  +0.104,Y -30.437,A +9.523,E1 -0.697,E3 +11.922,E4 +11.922} C_DIS
 LIN_REL {X  -0.181,Y -24.092,A +3.076,E1 -0.369,E3 +9.649,E4 +9.649} C_DIS
 LIN_REL {X  -0.102,Y -18.045,A -0.170,E1 +0.341,E3 +7.385,E4 +7.385} C_DIS
 LIN_REL {X  +0.326,Y -18.391,A -5.726,E1 +0.955,E3 +7.697,E4 +7.697} C_DIS
 LIN_REL {X  +0.491,Y -18.767,A +2.216,E1 +0.123,E3 +8.010,E4 +8.010} C_DIS
 LIN_REL {X  +0.467,Y -28.111,A +9.507,E1 -0.870,E3 +12.265,E4 +12.265} C_DIS
 LIN_REL {X  +0.039,Y -23.862,A +3.481,E1 -0.660,E3 +10.651,E4 +10.651} C_DIS
 LIN_REL {X  -0.570,Y -41.050,A -0.648,E1 -0.028,E3 +18.856,E4 +18.856} C_DIS
 LIN_REL {X  -0.534,Y -58.098,A +0.036,E1 +0.433,E3 +28.087,E4 +28.087} C_DIS
 LIN_REL {X  +0.144,Y -73.535,A +0.126,E1 -0.032,E3 +36.412,E4 +36.412} C_DIS
 LIN_REL {X  +0.037,Y -121.942,A +0.007,E1 -0.008,E3 +60.499,E4 +60.499} C_DIS
 LIN_REL {X  +0.019,Y -79.330,A -0.000,E1 -0.003,E3 +39.383,E4 +39.383} C_DIS
 LIN_REL {X  +0.245,Y -64.650,A +0.000,E1 -0.029,E3 +32.274,E4 +32.274} C_DIS
 LIN_REL {X  +1.899,Y -49.083,A +0.000,E1 -0.215,E3 +25.808,E4 +25.808} C_DIS
 LIN_REL {X  +5.378,Y -35.510,A +0.000,E1 -0.583,E3 +21.553,E4 +21.553} C_DIS
 LIN_REL {X  +5.642,Y -18.817,A +0.004,E1 -0.635,E3 +13.229,E4 +13.229} C_DIS
 LIN_REL {X  +7.917,Y -16.323,A +0.051,E1 -0.961,E3 +13.052,E4 +13.052} C_DIS
 LIN_REL {X  +12.018,Y -15.561,A +0.370,E1 -1.457,E3 +13.903,E4 +13.903} C_DIS
 LIN_REL {X  +10.570,Y -9.673,A +7.310,E1 -2.479,E3 +10.275,E4 +10.275} C_DIS
 LIN_REL {X  +4.255,Y -3.456,A +1.241,E1 -0.724,E3 +4.256,E4 +4.256} C_DIS
 LIN_REL {X  +11.408,Y -7.555,A +1.130,E1 -1.883,E3 +11.960,E4 +11.960} C_DIS
 LIN_REL {X  +12.962,Y -7.974,A +12.026,E1 -5.240,E3 +17.538,E4 +17.538} C_DIS
 LIN_REL {X  +7.148,Y -5.221,A +6.312,E1 -3.675,E3 +13.440,E4 +13.440} C_DIS
 LIN_REL {X  +9.468,Y -13.695,A +1.556,E1 -4.637,E3 +32.520,E4 +32.520} C_DIS
 LIN_REL {X  +4.887,Y -21.033,A +0.000,E1 -6.266,E3 +56.028,E4 +56.028} C_DIS
 LIN_REL {X  -1.582,Y -10.452,A +0.000,E1 -9.667,E3 +59.175,E4 +59.175} C_DIS
 LIN_REL {X  -1.996,Y +5.242,A +0.000,E1 -7.631,E3 +32.957,E4 +32.957} C_DIS
 LIN_REL {X  -1.206,Y +19.900,A +0.000,E1 -13.797,E3 +34.457,E4 +34.457} C_DIS
 LIN_REL {X  -8.415,Y +18.832,A +0.000,E1 -15.882,E3 +32.725,E4 +32.725} C_DIS
 LIN_REL {X  -15.399,Y +11.360,A +0.000,E1 -19.863,E3 +25.575,E4 +25.575} C_DIS
 LIN_REL {X  -8.440,Y +5.222,A +0.000,E1 -7.577,E3 +10.055,E4 +10.055} C_DIS
 LIN_REL {X  -11.339,Y +8.734,A +0.000,E1 -7.953,E3 +15.146,E4 +15.146} C_DIS
 LIN_REL {X  -16.013,Y +16.758,A +0.000,E1 -12.003,E3 +11.638,E4 +11.638} C_DIS
 LIN_REL {X  -9.636,Y +11.675,A +0.000,E1 -6.794,E3 +19.363,E4 +19.363} C_DIS
ENDFOR

HALT
END
